TYPE TcoAmsAddr : STRUCT
    netId : ARRAY[0..5] OF BYTE;
    port : WORD;
END_STRUCT
END_TYPE

(* stored: Version 1.1.0.1, ProductVersion 3.1.4024.9
   DUT TcoAmsAddr: Id {8e2bce8c-c380-0a15-1e45-9f0f577c1d6f} *)
